INTERFACE IJsonExtender EXTENDS TwinCAT_OpenFramework_Core.IObject

METHOD ExtendAtFinish
VAR_INPUT
	jsonSaxWriter : REFERENCE TO Tc3_JsonXml.FB_JsonSaxPrettyWriter;	
END_VAR
END_METHOD

METHOD ExtendAtStart
VAR_INPUT
	jsonSaxWriter : REFERENCE TO Tc3_JsonXml.FB_JsonSaxPrettyWriter;	
END_VAR
END_METHOD

END_INTERFACE

(* stored: Version 1.1.0.1
   Itf IJsonExtender: Id {4855e1bf-29d3-434d-ad18-57cfe564a05a}
   Method ExtendAtFinish: Id {3bd84534-1712-40b5-9503-1fc6ee164105}
   Method ExtendAtStart: Id {9509cef5-06c5-4632-a66c-dbe1c085047e} *)
